// Mitsubishi GX Works2 project: plc_first_test   PLC: Q03UDV

PROGRAM MAIN
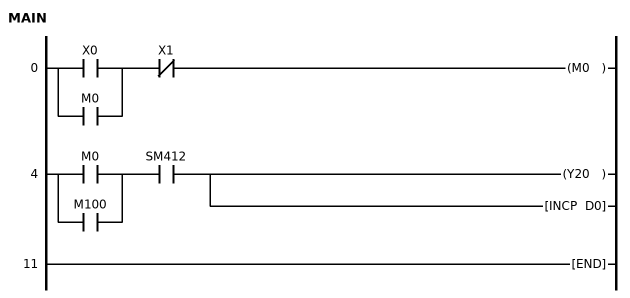
0     LD      X0
      OR      M0
      ANI     X1
      OUT     M0
4     LD      M0
      OR      M100
      AND     SM412
      OUT     Y20
      INCP    D0
11    END
END_PROGRAM
